TYPE ST_ADS_DFOIL :
(*************************************************************************************************)
(*  FILENAME:    ST_ADS_DFOIL                                                                    *)
(*  PROJECT:     CALMAR PUPLC                                                                    *)
(*  COPYRIGHT:   All rights reserved (c) Wifag//Polytype, Fribourg/Switzerland (2019)            *)
(*  ENVIRONMENT: TwinCAT PLC                                                                     *)
(*  VERSION:     <version>                                                                       *)
(*************************************************************************************************)
(*  DESCRIPTION:                                                                   <description> *)
(*    ADS structure dFoil system.                                                                *)
(*                                                                                </description> *)
(*************************************************************************************************)

STRUCT
  iO_Version         : INT    := 010000;  (*1.0.0*)
  aO_Type            : STRING := 'dFoil';
  aO_Name            : STRING := 'dFoil';

  bI_Enable          : BOOL := TRUE;      (*Enable this device*)
  iO_MaxNbRecords    : UINT  := SIZEOF(sI_dFoilUsagePos) / SIZEOF(sI_dFoilUsagePos[1]);

  iI_UsedNbRecords   : UINT;
  sI_dFoilUsagePos   : ARRAY[1..20] OF ST_DFOIL_RECORD;
END_STRUCT
END_TYPE

(* stored: Version 1.1.0.1, ProductVersion 3.1.4024.11
   DUT ST_ADS_DFOIL: Id {52ca6b52-98bc-4ab2-8c5b-de91f722c6e6} *)
